// TIA Portal project "S7-1500 Analog Giriş ile Seviye Ölçümü" (V18)

(* hardware
DEVICE "S7-1500/ET200MP station_1"  S7-1500 station
   slot 0: "Rail_0"  Rack  6ES7 590-1***0-0AA0
   slot 1: "PLC_1"  CPU 1512C-1 PN  6ES7 512-1CK01-0AB0  V2.8
      slot 3: "CPU display_1"  6ES7591-1AA00-0AA0
      slot 32768: "PROFINET interface_1"  X1
         slot 32769: "Port_1"  X1 P1
         slot 32770: "Port_2"  X1 P2
      slot 34817: "Virtual CP interface port_1"  Virtual CP interface port  Virtual CP interface port
*)

// ===== PLC "PLC_1"  CPU 1512C-1 PN =====

VAR_GLOBAL   // PLC tag table "Default tag table"
   "Otopark Dolu" AT %Q0.0 : Bool;
   "Reset" AT %I0.0 : Bool;
   "Arttır" AT %I0.1 : Bool;
   "Azalt" AT %I0.2 : Bool;
   "Uyarı" AT %M0.0 : Bool;
   "Araç Sayısı" AT %MW2 : Int;
   "Otopark Boş" AT %Q0.1 : Bool;
   "boş" AT %MW4 : Int;
   "Tag_1" AT %IW124 : Word;
   "Tag_2" AT %MW124 : Word;
   "Tag_3" AT %IW126 : Word;
   "Tag_4" AT %MW126 : Word;
   "Tag_5" AT %MD10 : DWord;
   "Tag_6" AT %MD20 : DWord;
END_VAR

ORGANIZATION_BLOCK "Main"   // OB1, LAD, ProgramCycle
TITLE = "Main Program Sweep (Cycle)"
{ S7_Optimized_Access := 'TRUE' }
VERSION : 0.1
   VAR_INPUT
      Initial_Call : Bool;   // Initial call of this OB
      Remanence : Bool;   // =True, if remanent data are available
   END_VAR
BEGIN

REGION Network 1
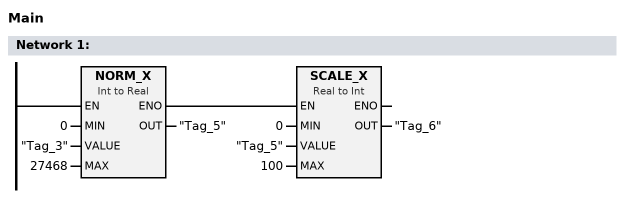
   RUNG wire#powerrail
      { S7_Templates := "[SrcType := Int, DestType := Real]" } Normalize(min := 0, value := "Tag_3", max := 27468, out => "Tag_5")
      { S7_Templates := "[SrcType := Real, DestType := Int]" } Scale(min := 0, value := "Tag_5", max := 100, out => "Tag_6")
   END_RUNG
   // the same network as SCL:
   "Tag_5" := NORM_X(MIN := 0, VALUE := "Tag_3", MAX := 27468);
   "Tag_6" := SCALE_X(MIN := 0, VALUE := "Tag_5", MAX := 100);
END_REGION
END_ORGANIZATION_BLOCK